// TIA Portal V20 export
TYPE "UDT_BoolEnable"
   STRUCT
      IsEnabled : Bool;
      Value : Bool;
   END_STRUCT;
END_TYPE
